(* IEC 61131-3 sources: eebus-docker-bridge/codesys, 12 files *)

(* ---- eAnlagenstatus.st ---- *)
// Betriebszustand der Anlage, den die Brücke an die Steuerbox meldet
// (FNN-Hinweis 4.1.2.7). Zahlenwerte identisch mit anlagenstatus* in anlage.go.
{attribute 'qualified_only'}
{attribute 'strict'}
TYPE eAnlagenstatus :
(
	Normal   := 0,
	Stoerung := 1,   // Anlage kann Grenzen nicht umsetzen
	Standby  := 2
) UINT;
END_TYPE

(* ---- eEebusVerbindung.st ---- *)
// Verbindungszustand zwischen Brücke und Steuerbox.
// Zahlenwerte identisch mit Verbindung in bruecke.go.
{attribute 'qualified_only'}
{attribute 'strict'}
TYPE eEebusVerbindung :
(
	KeinPartner := 0,    // kein SKI der Steuerbox konfiguriert
	Getrennt    := 1,
	Verbunden   := 2,
	Unbekannt   := 99
) UINT;
END_TYPE

(* ---- eLpcZustand.st ---- *)
// Zustand der Use Cases LPC (Bezug) und LPP (Einspeisung), wie ihn die
// EEBUS-Brücke meldet. Beide haben denselben Zustandsautomaten.
// Zahlenwerte identisch mit LpcZustand in bruecke.go.
{attribute 'qualified_only'}
{attribute 'strict'}
TYPE eLpcZustand :
(
	Init                := 0,   // nach Neustart, Failsafe-Grenze gilt
	UnbegrenztGesteuert := 1,   // Steuerbox verbunden, keine aktive Grenze
	Begrenzt            := 2,   // Grenze des Netzbetreibers aktiv
	Failsafe            := 3,   // Heartbeat ausgefallen, Failsafe-Grenze gilt
	UnbegrenztAutonom   := 4,   // keine Kommunikation, Failsafe-Mindestdauer abgelaufen
	Unbekannt           := 99   // Brücke nicht erreichbar oder Wert ungültig
) UINT;
END_TYPE

(* ---- ST_EebusMgcp.st ---- *)
// Messwerte am Netzanschlusspunkt für den Use Case MGCP (Monitoring of Grid
// Connection Point). Vorzeichen: Bezug aus dem Netz positiv, Einspeisung negativ.
// Ein Wert geht nur als gültig an die Steuerbox, wenn sein Bit in wGueltig
// gesetzt ist. Leistung und beide Energien sind Pflicht, Strom, Spannung,
// Frequenz und PV-Faktor je nach MGCP_MESSWERTE.
TYPE ST_EebusMgcp :
STRUCT
	diLeistungW           : DINT;                   // Bit 0
	ulEnergieEinspeisungWh: ULINT;                  // Bit 1, Zählerstand
	ulEnergieBezugWh      : ULINT;                  // Bit 2, Zählerstand
	aStromPhaseMA         : ARRAY [1..3] OF DINT;   // Bit 3..5, in mA
	aSpannungPhase01V     : ARRAY [1..3] OF UINT;   // Bit 6..8, in 0,1 V
	uiFrequenz001Hz       : UINT;                   // Bit 9, in 0,01 Hz
	uiPvFaktor01Prozent   : UINT;                   // Bit 10, PV-Einspeisebegrenzungsfaktor in 0,1 %
	wGueltig              : WORD;                   // Gültigkeitsbits wie oben
END_STRUCT
END_TYPE

(* ---- ST_EebusMpc.st ---- *)
// Messwerte der Anlage für den Use Case MPC (Monitoring of Power Consumption).
// Vorzeichen nach EEBUS: Bezug positiv, Erzeugung negativ.
// Ein Wert geht nur als gültig an die Steuerbox, wenn sein Bit in wGueltig
// gesetzt ist. Welche Werte die Brücke überhaupt anbietet, steht in
// MPC_MESSWERTE (Konfiguration des Containers).
TYPE ST_EebusMpc :
STRUCT
	diLeistungW         : DINT;                     // Bit 0
	aLeistungPhaseW     : ARRAY [1..3] OF DINT;     // Bit 1..3 (L1..L3)
	ulEnergieBezugWh    : ULINT;                    // Bit 4, Zählerstand
	ulEnergieErzeugungWh: ULINT;                    // Bit 5, Zählerstand
	aStromPhaseMA       : ARRAY [1..3] OF DINT;     // Bit 6..8, in mA
	aSpannungPhase01V   : ARRAY [1..3] OF UINT;     // Bit 9..11, in 0,1 V
	uiFrequenz001Hz     : UINT;                     // Bit 12, in 0,01 Hz
	wGueltig            : WORD;                     // Gültigkeitsbits wie oben
END_STRUCT
END_TYPE

(* ---- GvlEebus.st ---- *)
// Prozessabbild der Modbus-Verbindung zur EEBUS-Brücke (Erweiterungsversion 2).
// Mapping im Gerätebaum (Modbus TCP Client -> Server 127.0.0.1:5502):
//   Kanal 1: FC04 Read Input Registers,    Offset 0, Länge 31, Zyklus 200 ms -> aInputRegister
//   Kanal 2: FC16 Write Multiple Registers, Offset 0, Länge 61, Zyklus 1 s   -> aHoldingRegister
// Alle Holding-Register in EINEM Kanal schreiben: Dann sieht die Brücke immer
// einen zusammengehörigen Stand von Messwerten und Gültigkeitsmasken.
//
// Bestehende Projekte mit FbEebusLpc (14 Input-, 3 Holding-Register) laufen
// unverändert weiter, siehe FbEebusLpc.
{attribute 'qualified_only'}
VAR_GLOBAL
	aInputRegister   : ARRAY [0..30] OF WORD;   // Brücke -> SPS
	aHoldingRegister : ARRAY [0..60] OF WORD;   // SPS -> Brücke
END_VAR

(* ---- FuEebusRegister.st ---- *)
// Hilfsfunktionen: Werte in die Holding-Register der Brücke schreiben bzw.
// aus den Input-Registern lesen. Mehrwortige Werte: High-Word zuerst.

FUNCTION FuEebusSchreibeDint : BOOL
VAR_IN_OUT
	aRegister : ARRAY [0..60] OF WORD;
END_VAR
VAR_INPUT
	iIndex : INT;
	diWert : DINT;
END_VAR
VAR
	dwWert : DWORD;
END_VAR
dwWert := DINT_TO_DWORD(diWert);
aRegister[iIndex]     := DWORD_TO_WORD(SHR(dwWert, 16));
aRegister[iIndex + 1] := DWORD_TO_WORD(dwWert);
FuEebusSchreibeDint := TRUE;
END_FUNCTION

FUNCTION FuEebusSchreibeUdint : BOOL
VAR_IN_OUT
	aRegister : ARRAY [0..60] OF WORD;
END_VAR
VAR_INPUT
	iIndex  : INT;
	udiWert : UDINT;
END_VAR
aRegister[iIndex]     := UDINT_TO_WORD(SHR(udiWert, 16));
aRegister[iIndex + 1] := UDINT_TO_WORD(udiWert AND 16#0000FFFF);
FuEebusSchreibeUdint := TRUE;
END_FUNCTION

FUNCTION FuEebusSchreibeUlint : BOOL
VAR_IN_OUT
	aRegister : ARRAY [0..60] OF WORD;
END_VAR
VAR_INPUT
	iIndex : INT;
	ulWert : ULINT;
END_VAR
aRegister[iIndex]     := ULINT_TO_WORD(SHR(ulWert, 48));
aRegister[iIndex + 1] := ULINT_TO_WORD(SHR(ulWert, 32));
aRegister[iIndex + 2] := ULINT_TO_WORD(SHR(ulWert, 16));
aRegister[iIndex + 3] := ULINT_TO_WORD(ulWert);
FuEebusSchreibeUlint := TRUE;
END_FUNCTION

FUNCTION FuEebusLiesUdint : UDINT
VAR_IN_OUT
	aRegister : ARRAY [0..30] OF WORD;
END_VAR
VAR_INPUT
	iIndex : INT;
END_VAR
FuEebusLiesUdint := SHL(WORD_TO_UDINT(aRegister[iIndex]), 16) OR WORD_TO_UDINT(aRegister[iIndex + 1]);
END_FUNCTION

(* ---- FbEebusBegrenzung.st ---- *)
// Eine Richtung der Leistungsbegrenzung durch die Steuerbox:
//   iBasis := 2   Bezug (LPC, Paragraf 14a EnWG)
//   iBasis := 17  Einspeisung (LPP, Paragraf 9 EEG)
// Beide Blöcke der Input-Register sind gleich aufgebaut.
//
// Die Grenze bezieht sich laut FNN-Hinweis auf den Netzanschlusspunkt: Die
// Regelung muss sie dort einhalten (Messwert am Netzanschlusspunkt), nicht an
// einer einzelnen Last.
//
// Ist die Brücke ausgefallen oder bietet sie den Use Case nicht an, gilt die
// lokale Ersatzgrenze (sichere Seite, wie im Failsafe).
FUNCTION_BLOCK FbEebusBegrenzung
VAR_INPUT
	xBrueckeOk       : BOOL;                     // von FbEebusBruecke
	xUseCaseAktiv    : BOOL;                     // von FbEebusBruecke (xLpcAktiv bzw. xLppAktiv)
	iBasis           : INT := 2;                 // 2 = Bezug, 17 = Einspeisung
	udiErsatzgrenzeW : UDINT := 4200;            // gilt, solange die Brücke nicht verfügbar ist
END_VAR
VAR_IN_OUT
	aInputRegister   : ARRAY [0..30] OF WORD;
END_VAR
VAR_OUTPUT
	xBegrenzungAktiv    : BOOL;                  // udiLeistungsgrenzeW muss eingehalten werden
	udiLeistungsgrenzeW : UDINT;                 // nur gültig bei xBegrenzungAktiv
	eZustand            : eLpcZustand;
	udiRestdauerS       : UDINT;                 // Restlaufzeit der Grenze, 0 = unbefristet
	udiGrenzeNetzW      : UDINT;                 // zuletzt empfangene Grenze (Diagnose)
	udiFailsafeGrenzeW  : UDINT;                 // aktuelle Failsafe-Grenze (Diagnose)
	xErsatzgrenze       : BOOL;                  // Ersatzgrenze aktiv, Brücke nicht verfügbar
END_VAR
VAR
	uiRohZustand : UINT;
END_VAR
VAR CONSTANT
	// Offsets im Block, identisch mit blk* in modbus.go
	iBlkZustand          : INT := 0;
	iBlkWirksameGrenze   : INT := 2;
	iBlkBegrenzungAktiv  : INT := 4;
	iBlkGrenzeNetz       : INT := 5;
	iBlkRestdauer        : INT := 7;
	iBlkFailsafeGrenze   : INT := 9;
END_VAR

uiRohZustand := WORD_TO_UINT(aInputRegister[iBasis + iBlkZustand]);

IF xBrueckeOk AND xUseCaseAktiv AND uiRohZustand <= 4 THEN
	CASE uiRohZustand OF
		0: eZustand := eLpcZustand.Init;
		1: eZustand := eLpcZustand.UnbegrenztGesteuert;
		2: eZustand := eLpcZustand.Begrenzt;
		3: eZustand := eLpcZustand.Failsafe;
		4: eZustand := eLpcZustand.UnbegrenztAutonom;
	END_CASE
	xBegrenzungAktiv    := aInputRegister[iBasis + iBlkBegrenzungAktiv] <> 0;
	udiLeistungsgrenzeW := FuEebusLiesUdint(aRegister := aInputRegister, iIndex := iBasis + iBlkWirksameGrenze);
	udiRestdauerS       := FuEebusLiesUdint(aRegister := aInputRegister, iIndex := iBasis + iBlkRestdauer);
	udiGrenzeNetzW      := FuEebusLiesUdint(aRegister := aInputRegister, iIndex := iBasis + iBlkGrenzeNetz);
	udiFailsafeGrenzeW  := FuEebusLiesUdint(aRegister := aInputRegister, iIndex := iBasis + iBlkFailsafeGrenze);
	xErsatzgrenze       := FALSE;
ELSE
	// Zustand der Steuerbox unbekannt: wie Failsafe verhalten
	eZustand            := eLpcZustand.Unbekannt;
	xBegrenzungAktiv    := TRUE;
	udiLeistungsgrenzeW := udiErsatzgrenzeW;
	udiRestdauerS       := 0;
	udiGrenzeNetzW      := 0;
	udiFailsafeGrenzeW  := udiErsatzgrenzeW;
	xErsatzgrenze       := TRUE;
END_IF
END_FUNCTION_BLOCK

(* ---- FbEebusBruecke.st ---- *)
// Verbindung zur EEBUS-Brücke (Erweiterungsversion 2: LPC, LPP, MPC, MGCP).
//
// Der Baustein
// - überwacht Lebenszeichen und Schnittstellenversion der Brücke,
// - dekodiert Verbindung, Heartbeat und die Use-Case-Masken,
// - schreibt SPS-Lebenszeichen, Nennleistungen und Anlagenstatus in die
//   Holding-Register (Register 0 bis 4 und 7).
//
// Die Begrenzungen je Richtung wertet FbEebusBegrenzung aus, die Messwerte
// schreibt FbEebusMesswerte. Alle drei arbeiten auf denselben Registerabbildern.
FUNCTION_BLOCK FbEebusBruecke
VAR_INPUT
	xFreigabe                 : BOOL;            // Auswertung aktiv
	udiNennleistungBezugW     : UDINT;           // max. Leistungsaufnahme der Anlage in W (LPC), 0 = Vorgabe der Brücke
	udiNennleistungErzeugungW : UDINT;           // max. Einspeiseleistung in W (LPP), 0 = Vorgabe der Brücke
	eStatus                   : eAnlagenstatus;  // Störung der Anlage an die Steuerbox melden
	tBrueckeTimeout           : TIME := T#10S;   // max. Zeit ohne Änderung des Brücken-Lebenszeichens
END_VAR
VAR_IN_OUT
	aInputRegister   : ARRAY [0..30] OF WORD;    // Abbild der Input-Register der Brücke
	aHoldingRegister : ARRAY [0..60] OF WORD;    // an die Brücke zu schreibende Register
END_VAR
VAR_OUTPUT
	xBrueckeOk          : BOOL;                  // Brücke lebt und Version passt
	eVerbindung         : eEebusVerbindung;
	uiHeartbeatAlterS   : UINT;                  // Sekunden seit letztem Heartbeat der Steuerbox, 65535 = nie
	xLpcAktiv           : BOOL;                  // Use Case von der Brücke angeboten ...
	xLppAktiv           : BOOL;
	xMpcAktiv           : BOOL;
	xMgcpAktiv          : BOOL;
	wUseCasesSteuerbox  : WORD;                  // ... und von der Steuerbox unterstützt (Bits wie wUseCases*)
	udiFailsafeMindestdauerS : UDINT;            // gemeinsam für LPC und LPP
	xFehler             : BOOL;
	udiFehlerId         : UDINT;                 // siehe Konstanten udiFehler*
END_VAR
VAR
	wLebenszeichenAlt   : WORD;
	tonBrueckeTimeout   : TON;
	tonSekundentakt     : TON;
	uiLebenszeichenSps  : UINT;
	xVersionOk          : BOOL;
	wUseCases           : WORD;
END_VAR
VAR CONSTANT
	uiSchnittstellenVersion : UINT := 1;   // SchnittstellenVersion in modbus.go
	uiErweiterungMindestens : UINT := 2;   // ErweiterungsVersion in modbus.go

	// Input-Register, identisch mit modbus.go
	iRegLebenszeichen       : INT := 0;
	iRegVersion             : INT := 1;
	iRegVerbindung          : INT := 3;
	iRegHeartbeatAlter      : INT := 13;
	iRegErweiterung         : INT := 14;
	iRegUseCasesLokal       : INT := 15;
	iRegUseCasesSteuerbox   : INT := 16;
	iRegMindestdauer        : INT := 29;

	// Holding-Register, identisch mit modbus.go
	iRegSpsLebenszeichen    : INT := 0;
	iRegNennleistung        : INT := 1;
	iRegNennleistungErzeugung : INT := 3;
	iRegAnlagenstatus       : INT := 7;

	// Bits der Use-Case-Masken
	wUseCaseLpc             : WORD := 16#0001;
	wUseCaseLpp             : WORD := 16#0002;
	wUseCaseMpc             : WORD := 16#0004;
	wUseCaseMgcp            : WORD := 16#0008;

	// Fehlernummern
	udiFehlerKeine          : UDINT := 0;
	udiFehlerBrueckeTimeout : UDINT := 1;   // Lebenszeichen der Brücke steht
	udiFehlerVersion        : UDINT := 2;   // Registerlayout passt nicht (Brücke zu alt?)
END_VAR

// ---------------------------------------------------------------------------
// Register an die Brücke
// ---------------------------------------------------------------------------
tonSekundentakt(IN := NOT tonSekundentakt.Q, PT := T#1S);
IF tonSekundentakt.Q THEN
	uiLebenszeichenSps := uiLebenszeichenSps + 1;   // Überlauf ist gewollt
END_IF

aHoldingRegister[iRegSpsLebenszeichen] := UINT_TO_WORD(uiLebenszeichenSps);
FuEebusSchreibeUdint(aRegister := aHoldingRegister, iIndex := iRegNennleistung, udiWert := udiNennleistungBezugW);
FuEebusSchreibeUdint(aRegister := aHoldingRegister, iIndex := iRegNennleistungErzeugung, udiWert := udiNennleistungErzeugungW);
aHoldingRegister[iRegAnlagenstatus] := TO_WORD(eStatus);

// ---------------------------------------------------------------------------
// Überwachung der Brücke
// ---------------------------------------------------------------------------
tonBrueckeTimeout(IN := xFreigabe AND (aInputRegister[iRegLebenszeichen] = wLebenszeichenAlt),
                  PT := tBrueckeTimeout);
wLebenszeichenAlt := aInputRegister[iRegLebenszeichen];

xVersionOk := WORD_TO_UINT(aInputRegister[iRegVersion]) = uiSchnittstellenVersion
              AND WORD_TO_UINT(aInputRegister[iRegErweiterung]) >= uiErweiterungMindestens;
xBrueckeOk := xFreigabe AND NOT tonBrueckeTimeout.Q AND xVersionOk;

IF xBrueckeOk THEN
	CASE WORD_TO_UINT(aInputRegister[iRegVerbindung]) OF
		0: eVerbindung := eEebusVerbindung.KeinPartner;
		1: eVerbindung := eEebusVerbindung.Getrennt;
		2: eVerbindung := eEebusVerbindung.Verbunden;
	ELSE
		eVerbindung := eEebusVerbindung.Unbekannt;
	END_CASE
	uiHeartbeatAlterS        := WORD_TO_UINT(aInputRegister[iRegHeartbeatAlter]);
	wUseCases                := aInputRegister[iRegUseCasesLokal];
	wUseCasesSteuerbox       := aInputRegister[iRegUseCasesSteuerbox];
	udiFailsafeMindestdauerS := FuEebusLiesUdint(aRegister := aInputRegister, iIndex := iRegMindestdauer);
	xFehler                  := FALSE;
	udiFehlerId              := udiFehlerKeine;
ELSE
	eVerbindung              := eEebusVerbindung.Unbekannt;
	uiHeartbeatAlterS        := 16#FFFF;
	wUseCases                := 0;
	wUseCasesSteuerbox       := 0;
	udiFailsafeMindestdauerS := 0;
	xFehler                  := xFreigabe;
	IF NOT xFreigabe THEN
		udiFehlerId := udiFehlerKeine;
	ELSIF tonBrueckeTimeout.Q THEN
		udiFehlerId := udiFehlerBrueckeTimeout;
	ELSE
		udiFehlerId := udiFehlerVersion;
	END_IF
END_IF

xLpcAktiv  := (wUseCases AND wUseCaseLpc) <> 0;
xLppAktiv  := (wUseCases AND wUseCaseLpp) <> 0;
xMpcAktiv  := (wUseCases AND wUseCaseMpc) <> 0;
xMgcpAktiv := (wUseCases AND wUseCaseMgcp) <> 0;
END_FUNCTION_BLOCK

(* ---- FbEebusLpc.st ---- *)
// Auswertung der EEBUS-LPC-Brücke (Docker-Container auf derselben Steuerung).
//
// VERALTET: Für neue Projekte FbEebusBruecke, FbEebusBegrenzung und
// FbEebusMesswerte verwenden (LPP, Messwerte, Anlagenstatus). Dieser Baustein
// läuft mit neueren Brücken unverändert weiter, weil die Register 0 bis 13
// und 0 bis 2 gleich geblieben sind (Schnittstellenversion 1).
//
// Die Brücke liefert die vom Netzbetreiber vorgegebene Leistungsgrenze
// (Use Case LPC, Paragraf 14a EnWG) als Modbus-Input-Register. Der Baustein
// - überwacht das Lebenszeichen und die Schnittstellenversion der Brücke,
// - dekodiert Zustand, Verbindung und wirksame Leistungsgrenze,
// - fällt bei Ausfall der Brücke auf eine lokale Ersatzgrenze zurück (sichere Seite),
// - erzeugt die Holding-Register (SPS-Lebenszeichen, Nennleistung) für die Brücke.
//
// Der Baustein greift auf keine globalen Variablen zu. Die Kopplung an das
// Modbus-Prozessabbild erfolgt beim Aufruf.
FUNCTION_BLOCK FbEebusLpc
VAR_INPUT
	xFreigabe           : BOOL;                    // Auswertung aktiv
	aInputRegister      : ARRAY [0..13] OF WORD;   // Abbild der Input-Register der Brücke
	udiNennleistungMaxW : UDINT;                   // max. Leistungsaufnahme der Anlage in W, wird an die Steuerbox gemeldet
	udiErsatzgrenzeW    : UDINT := 4200;           // gilt, solange die Brücke nicht verfügbar ist
	tBrueckeTimeout     : TIME := T#10S;           // max. Zeit ohne Änderung des Brücken-Lebenszeichens
END_VAR
VAR_OUTPUT
	xBrueckeOk          : BOOL;                    // Brücke lebt und Schnittstellenversion passt
	xBegrenzungAktiv    : BOOL;                    // udiLeistungsgrenzeW muss eingehalten werden
	udiLeistungsgrenzeW : UDINT;                   // nur gültig bei xBegrenzungAktiv
	eZustand            : eLpcZustand;
	eVerbindung         : eEebusVerbindung;
	udiRestdauerS       : UDINT;                   // Restlaufzeit der Grenze, 0 = unbefristet
	uiHeartbeatAlterS   : UINT;                    // Sekunden seit letztem Heartbeat der Steuerbox
	xFehler             : BOOL;
	udiFehlerId         : UDINT;                   // siehe Konstanten udiFehler*
	aHoldingRegister    : ARRAY [0..2] OF WORD;    // an die Brücke zu schreibende Register
END_VAR
VAR
	wLebenszeichenAlt   : WORD;
	tonBrueckeTimeout   : TON;
	tonSekundentakt     : TON;
	uiLebenszeichenSps  : UINT;
	uiRohZustand        : UINT;
	uiRohVerbindung     : UINT;
	xVersionOk          : BOOL;
	xZustandGueltig     : BOOL;
END_VAR
VAR CONSTANT
	uiSchnittstellenVersion   : UINT := 1;         // muss zu SchnittstellenVersion in modbus.go passen

	// Input-Register, identisch mit modbus.go
	iRegLebenszeichen         : INT := 0;
	iRegVersion               : INT := 1;
	iRegZustand               : INT := 2;
	iRegVerbindung            : INT := 3;
	iRegWirksameGrenzeHi      : INT := 4;
	iRegWirksameGrenzeLo      : INT := 5;
	iRegBegrenzungAktiv       : INT := 6;
	iRegRestdauerHi           : INT := 9;
	iRegRestdauerLo           : INT := 10;
	iRegHeartbeatAlter        : INT := 13;

	// Holding-Register, identisch mit modbus.go
	iRegSpsLebenszeichen      : INT := 0;
	iRegNennleistungHi        : INT := 1;
	iRegNennleistungLo        : INT := 2;

	// Fehlernummern
	udiFehlerKeine            : UDINT := 0;
	udiFehlerBrueckeTimeout   : UDINT := 1;    // Lebenszeichen der Brücke steht
	udiFehlerVersion          : UDINT := 2;    // Registerlayout passt nicht
	udiFehlerZustandUngueltig : UDINT := 3;    // unbekannter Zustandswert
END_VAR

// ---------------------------------------------------------------------------
// Register an die Brücke: Lebenszeichen im Sekundentakt und Nennleistung
// ---------------------------------------------------------------------------
tonSekundentakt(IN := NOT tonSekundentakt.Q, PT := T#1S);
IF tonSekundentakt.Q THEN
	uiLebenszeichenSps := uiLebenszeichenSps + 1;   // Überlauf ist gewollt
END_IF

aHoldingRegister[iRegSpsLebenszeichen] := UINT_TO_WORD(uiLebenszeichenSps);
aHoldingRegister[iRegNennleistungHi]   := UDINT_TO_WORD(SHR(udiNennleistungMaxW, 16));
aHoldingRegister[iRegNennleistungLo]   := UDINT_TO_WORD(udiNennleistungMaxW AND 16#0000FFFF);

// ---------------------------------------------------------------------------
// Überwachung der Brücke
// ---------------------------------------------------------------------------
tonBrueckeTimeout(IN := xFreigabe AND (aInputRegister[iRegLebenszeichen] = wLebenszeichenAlt),
                  PT := tBrueckeTimeout);
wLebenszeichenAlt := aInputRegister[iRegLebenszeichen];

uiRohZustand    := WORD_TO_UINT(aInputRegister[iRegZustand]);
uiRohVerbindung := WORD_TO_UINT(aInputRegister[iRegVerbindung]);
xVersionOk      := WORD_TO_UINT(aInputRegister[iRegVersion]) = uiSchnittstellenVersion;
xZustandGueltig := uiRohZustand <= 4;

xBrueckeOk := xFreigabe AND NOT tonBrueckeTimeout.Q AND xVersionOk AND xZustandGueltig;

// ---------------------------------------------------------------------------
// Auswertung
// ---------------------------------------------------------------------------
IF NOT xFreigabe THEN
	xBegrenzungAktiv    := FALSE;
	udiLeistungsgrenzeW := 0;
	eZustand            := eLpcZustand.Unbekannt;
	eVerbindung         := eEebusVerbindung.Unbekannt;
	udiRestdauerS       := 0;
	uiHeartbeatAlterS   := 0;
	xFehler             := FALSE;
	udiFehlerId         := udiFehlerKeine;

ELSIF xBrueckeOk THEN
	CASE uiRohZustand OF
		0: eZustand := eLpcZustand.Init;
		1: eZustand := eLpcZustand.UnbegrenztGesteuert;
		2: eZustand := eLpcZustand.Begrenzt;
		3: eZustand := eLpcZustand.Failsafe;
		4: eZustand := eLpcZustand.UnbegrenztAutonom;
	ELSE
		eZustand := eLpcZustand.Unbekannt;
	END_CASE

	CASE uiRohVerbindung OF
		0: eVerbindung := eEebusVerbindung.KeinPartner;
		1: eVerbindung := eEebusVerbindung.Getrennt;
		2: eVerbindung := eEebusVerbindung.Verbunden;
	ELSE
		eVerbindung := eEebusVerbindung.Unbekannt;
	END_CASE

	xBegrenzungAktiv    := aInputRegister[iRegBegrenzungAktiv] <> 0;
	udiLeistungsgrenzeW := SHL(WORD_TO_UDINT(aInputRegister[iRegWirksameGrenzeHi]), 16)
	                       OR WORD_TO_UDINT(aInputRegister[iRegWirksameGrenzeLo]);
	udiRestdauerS       := SHL(WORD_TO_UDINT(aInputRegister[iRegRestdauerHi]), 16)
	                       OR WORD_TO_UDINT(aInputRegister[iRegRestdauerLo]);
	uiHeartbeatAlterS   := WORD_TO_UINT(aInputRegister[iRegHeartbeatAlter]);
	xFehler             := FALSE;
	udiFehlerId         := udiFehlerKeine;

ELSE
	// Brücke ausgefallen oder inkompatibel: Zustand der Steuerbox unbekannt,
	// daher wie Failsafe verhalten und die lokale Ersatzgrenze einhalten.
	xBegrenzungAktiv    := TRUE;
	udiLeistungsgrenzeW := udiErsatzgrenzeW;
	eZustand            := eLpcZustand.Unbekannt;
	eVerbindung         := eEebusVerbindung.Unbekannt;
	udiRestdauerS       := 0;
	uiHeartbeatAlterS   := 16#FFFF;
	xFehler             := TRUE;

	IF tonBrueckeTimeout.Q THEN
		udiFehlerId := udiFehlerBrueckeTimeout;
	ELSIF NOT xVersionOk THEN
		udiFehlerId := udiFehlerVersion;
	ELSE
		udiFehlerId := udiFehlerZustandUngueltig;
	END_IF
END_IF
END_FUNCTION_BLOCK

(* ---- FbEebusMesswerte.st ---- *)
// Schreibt die Messwerte für MPC (Anlage) und MGCP (Netzanschlusspunkt) in
// die Holding-Register 5 bis 60 der Brücke. Welche Werte die Brücke an die
// Steuerbox weitergibt, steht in ihrer Konfiguration (MPC_MESSWERTE,
// MGCP_MESSWERTE); ob ein Wert gerade gültig ist, in wGueltig der Strukturen.
//
// Mindestens die aktuelle Wirkleistung der Anlage muss die Steuerbox abfragen
// können (FNN-Hinweis 4.1.2.3). Ohne gültigen Wert meldet die Brücke ihn als
// ungültig.
FUNCTION_BLOCK FbEebusMesswerte
VAR_INPUT
	stMpc  : ST_EebusMpc;
	stMgcp : ST_EebusMgcp;
END_VAR
VAR_IN_OUT
	aHoldingRegister : ARRAY [0..60] OF WORD;
END_VAR
VAR
	i : INT;
END_VAR
VAR CONSTANT
	// Holding-Register, identisch mit modbus.go
	iRegMpcMaske        : INT := 5;
	iRegMgcpMaske       : INT := 6;
	iRegMpcP            : INT := 8;
	iRegMpcPL1          : INT := 10;
	iRegMpcEBezug       : INT := 16;
	iRegMpcEErzeugung   : INT := 20;
	iRegMpcIL1          : INT := 24;
	iRegMpcUL1          : INT := 30;
	iRegMpcF            : INT := 33;
	iRegMgcpP           : INT := 40;
	iRegMgcpEEinspeisung: INT := 42;
	iRegMgcpEBezug      : INT := 46;
	iRegMgcpIL1         : INT := 50;
	iRegMgcpUL1         : INT := 56;
	iRegMgcpF           : INT := 59;
	iRegMgcpPvFaktor    : INT := 60;
END_VAR

aHoldingRegister[iRegMpcMaske]  := stMpc.wGueltig;
aHoldingRegister[iRegMgcpMaske] := stMgcp.wGueltig;

// MPC
FuEebusSchreibeDint(aRegister := aHoldingRegister, iIndex := iRegMpcP, diWert := stMpc.diLeistungW);
FuEebusSchreibeUlint(aRegister := aHoldingRegister, iIndex := iRegMpcEBezug, ulWert := stMpc.ulEnergieBezugWh);
FuEebusSchreibeUlint(aRegister := aHoldingRegister, iIndex := iRegMpcEErzeugung, ulWert := stMpc.ulEnergieErzeugungWh);
aHoldingRegister[iRegMpcF] := UINT_TO_WORD(stMpc.uiFrequenz001Hz);
FOR i := 1 TO 3 DO
	FuEebusSchreibeDint(aRegister := aHoldingRegister, iIndex := iRegMpcPL1 + 2 * (i - 1), diWert := stMpc.aLeistungPhaseW[i]);
	FuEebusSchreibeDint(aRegister := aHoldingRegister, iIndex := iRegMpcIL1 + 2 * (i - 1), diWert := stMpc.aStromPhaseMA[i]);
	aHoldingRegister[iRegMpcUL1 + i - 1] := UINT_TO_WORD(stMpc.aSpannungPhase01V[i]);
END_FOR

// MGCP
FuEebusSchreibeDint(aRegister := aHoldingRegister, iIndex := iRegMgcpP, diWert := stMgcp.diLeistungW);
FuEebusSchreibeUlint(aRegister := aHoldingRegister, iIndex := iRegMgcpEEinspeisung, ulWert := stMgcp.ulEnergieEinspeisungWh);
FuEebusSchreibeUlint(aRegister := aHoldingRegister, iIndex := iRegMgcpEBezug, ulWert := stMgcp.ulEnergieBezugWh);
aHoldingRegister[iRegMgcpF]        := UINT_TO_WORD(stMgcp.uiFrequenz001Hz);
aHoldingRegister[iRegMgcpPvFaktor] := UINT_TO_WORD(stMgcp.uiPvFaktor01Prozent);
FOR i := 1 TO 3 DO
	FuEebusSchreibeDint(aRegister := aHoldingRegister, iIndex := iRegMgcpIL1 + 2 * (i - 1), diWert := stMgcp.aStromPhaseMA[i]);
	aHoldingRegister[iRegMgcpUL1 + i - 1] := UINT_TO_WORD(stMgcp.aSpannungPhase01V[i]);
END_FOR
END_FUNCTION_BLOCK

(* ---- PrgEnergiemanagement.st ---- *)
// Beispielaufruf mit allen Use Cases (Erweiterungsversion 2). Die Aufteilung
// der Grenzen auf die einzelnen Verbraucher und Erzeuger (Wallboxen,
// Wärmepumpe, PV-Wechselrichter, Speicher, ...) ist anlagenspezifisch.
//
// Wichtig (FNN-Hinweis, Fußnote 4): Die Grenzen beziehen sich auf den
// Netzanschlusspunkt. Die Regelung muss sie am Zähler des Netzanschlusspunkts
// einhalten. Bei einem EMS ist außerdem die Mindestbezugsleistung nach BNetzA
// BK6-22-300 Anlage 1 zu berücksichtigen.
PROGRAM PrgEnergiemanagement
VAR
	fbBruecke     : FbEebusBruecke;
	fbBezug       : FbEebusBegrenzung;
	fbEinspeisung : FbEebusBegrenzung;
	fbMesswerte   : FbEebusMesswerte;

	stMpc  : ST_EebusMpc;    // aus der Messung der steuerbaren Anlage füllen
	stMgcp : ST_EebusMgcp;   // aus dem Zähler am Netzanschlusspunkt füllen

	diNetzleistungW          : DINT;    // Messwert am Netzanschlusspunkt, Bezug positiv
	udiAnforderungW          : UDINT;   // ungeregelte Summenanforderung der steuerbaren Verbraucher
	udiFreigegebeneLeistungW : UDINT;   // Vorgabe an die Verteillogik
	udiPvSollW               : UDINT;   // Vorgabe an die PV-Wechselrichter
	udiPvMaxW                : UDINT := 8000;
	xAnlagenstoerung         : BOOL;
END_VAR

fbBruecke(
	xFreigabe                 := TRUE,
	udiNennleistungBezugW     := 22000,
	udiNennleistungErzeugungW := udiPvMaxW,
	eStatus                   := SEL(xAnlagenstoerung, eAnlagenstatus.Normal, eAnlagenstatus.Stoerung),
	tBrueckeTimeout           := T#10S,
	aInputRegister            := GvlEebus.aInputRegister,
	aHoldingRegister          := GvlEebus.aHoldingRegister);

fbBezug(
	xBrueckeOk       := fbBruecke.xBrueckeOk,
	xUseCaseAktiv    := fbBruecke.xLpcAktiv,
	iBasis           := 2,
	udiErsatzgrenzeW := 4200,
	aInputRegister   := GvlEebus.aInputRegister);

fbEinspeisung(
	xBrueckeOk       := fbBruecke.xBrueckeOk,
	xUseCaseAktiv    := fbBruecke.xLppAktiv,
	iBasis           := 17,
	udiErsatzgrenzeW := udiPvMaxW * 6 / 10,   // z. B. 60 % nach Netzanschlussvertrag
	aInputRegister   := GvlEebus.aInputRegister);

// Messwerte: hier nur die Netzleistung als Beispiel, alle Bits nur für
// tatsächlich gemessene Werte setzen.
stMgcp.diLeistungW := diNetzleistungW;
stMgcp.wGueltig    := 16#0001;
stMpc.diLeistungW  := UDINT_TO_DINT(udiFreigegebeneLeistungW);
stMpc.wGueltig     := 16#0001;
fbMesswerte(stMpc := stMpc, stMgcp := stMgcp, aHoldingRegister := GvlEebus.aHoldingRegister);

// Bezug begrenzen
IF fbBezug.xBegrenzungAktiv THEN
	udiFreigegebeneLeistungW := MIN(udiAnforderungW, fbBezug.udiLeistungsgrenzeW);
ELSE
	udiFreigegebeneLeistungW := udiAnforderungW;
END_IF

// Einspeisung begrenzen (vereinfacht: ohne Eigenverbrauch)
IF fbEinspeisung.xBegrenzungAktiv THEN
	udiPvSollW := MIN(udiPvMaxW, fbEinspeisung.udiLeistungsgrenzeW);
ELSE
	udiPvSollW := udiPvMaxW;
END_IF
END_PROGRAM
